FUNCTION ASSEMBLE_WORD_FROM_BYTES (* this Function combines the 2 BYTES to a WORD *)
  (* Standard: 61499-1; Description: Copyright (c) 2024 HR Agrartechnik GmbH This program and the accompanying materials are made available under the terms of the Eclipse Public License 2.0 which is available at https://www.eclipse.org/legal/epl-2.0/ SPDX-License-Identifier: EPL-2.0 *)
  (* Version 3.0, 2025-04-14, Patrick Aigner, changed package *)
  (* Version 1.1, 2024-07-28, Moritz Ortmeier, HR Agrartechnik, rename Function and change Input/Output Variables *)
  (* Version 1.0, 2024-02-22, Franz Höpfinger, HR Agrartechnik, initial Implementation *)
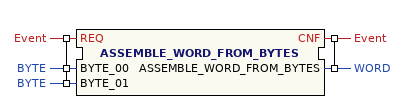
  EVENT_INPUT
    REQ WITH BYTE_00, BYTE_01;
  END_EVENT
  EVENT_OUTPUT
    CNF WITH ASSEMBLE_WORD_FROM_BYTES;
  END_EVENT
  VAR_INPUT
    BYTE_00 : BYTE;
    BYTE_01 : BYTE;
  END_VAR
  VAR_OUTPUT
    ASSEMBLE_WORD_FROM_BYTES : WORD;
  END_VAR
  BODY IN ST:
(* this Function combines the 2 BYTES to a WORD *)
FUNCTION ASSEMBLE_WORD_FROM_BYTES : WORD

VAR_INPUT
	BYTE_00 : BYTE;
	BYTE_01 : BYTE;
END_VAR

ASSEMBLE_WORD_FROM_BYTES.%B0 := BYTE_00;
ASSEMBLE_WORD_FROM_BYTES.%B1 := BYTE_01;

END_FUNCTION
  END_BODY
END_FUNCTION
